# EPICS substitutions: ioc/PSCApp/Db/devPSC.substitutions
file db/devPSC.db {
    pattern {AI_INDEX}
        {"0"}
        {"1"}
        {"2"}
        {"3"}
}
file db/devPSC.db {
    pattern {AO_INDEX}
        {"0"}
}
file db/devPSC.db {
    pattern {DI_INDEX}
        {"0"}
}
file db/devPSC.db {
    pattern {DO_INDEX}
        {"0"}
}
